// TIA Portal V17 export
// export: Created 2022-03-12T16:05:33.0426509Z, ExportSetting WithDefaults, DisplayName Totally Integrated Automation Portal, DisplayVersion V17, DisplayName TIA Portal Openness, DisplayVersion V17, DisplayName TIA Portal Version Control Interface, DisplayVersion V17, DisplayName STEP 7 Professional, DisplayVersion V17, DisplayName STEP 7 Safety, DisplayVersion V17, DisplayName WinCC Advanced / Unified PC, DisplayVersion V17
TYPE "CPG_typePackML_ModuleSts"
// stored: IsFailsafeCompliant false
   STRUCT
      cmd_Reset : Bool;   // Reset
      sts_Resetting_SC : Bool;   // Resetting State Complete
      cmd_Start : Bool;   // Start
      sts_Starting_SC : Bool;   // Starting State Complete
      cmd_Stop : Bool;   // Stop
      sts_Stopping_SC : Bool;   // Stopping State Complete
      cmd_Hold : Bool;   // Hold
      sts_Holding_SC : Bool;   // Holding State Complete
      cmd_UnHold : Bool;   // UnHold
      sts_UnHolding_SC : Bool;   // UnHolding State Complete
      cmd_Suspend : Bool;   // Suspend
      sts_Suspending_SC : Bool;   // Suspending State Complete
      cmd_UnSuspend : Bool;   // UnSuspend
      sts_UnSuspending_SC : Bool;   // UnSuspending State Complete
      cmd_Abort : Bool;   // Abort
      sts_Aborting_SC : Bool;   // Aborting State Complete
      cmd_Clear : Bool;   // Clear
      sts_Clearing_SC : Bool;   // Clearing State Complete
      sts_Execute_SC : Bool;   // Execute State Complete
      sts_Completing_SC : Bool;   // Completing State Complete
      moduleActive : Bool;   // Module Active Bit
      ONS : Bool;   // Internal One Shot Bit - Do not modify
   END_STRUCT;
END_TYPE
